(* PLC project VendorEdgeCases, RobotCo Vendor Edge Cases 1.0 *)
(* stored: creationDateTime 2026-05-30T00:00:00, modificationDateTime 2026-05-30T00:00:00 *)

PROGRAM VendorEdgeCases
  VAR
    A : INT := 1;
  END_VAR

            A := A + 1;
            A := A + 2;
          
END_PROGRAM
